Staubli VAL3: goTo.pgx

public program goTo(tool x_tTool, mdesc x_mDesc, num x_nMoveType, bool& x_bUnreached[], num x_nIndex)
  local point l_pTrsf
  local bool l_bInside
  local tool l_tTool
  local point l_pHere
  local string l_sMessage
  local num l_nSize
  local num i
  local mdesc l_mSpeed
  local joint l_jHere
  local joint l_jJoint
begin
  // the maximum size
  call getSizeItem(false,l_nSize)
  // get the trsf
  call getPoint(pToGo,false,x_nIndex)
  // check if the point is ok
  if pointToJoint(x_tTool,herej(),pToGo,l_jJoint)
    // step by step motion
    if x_nMoveType==0
      // or is not in range
      movej(pToGo,x_tTool,x_mDesc)
    else
      movel(pToGo,x_tTool,x_mDesc)
    endIf
  else
    // get the message point is not reachable
    call language:message(l_sMessage,-5)
    call use:type(0,12,"!!! "+l_sMessage)
  endIf
end
